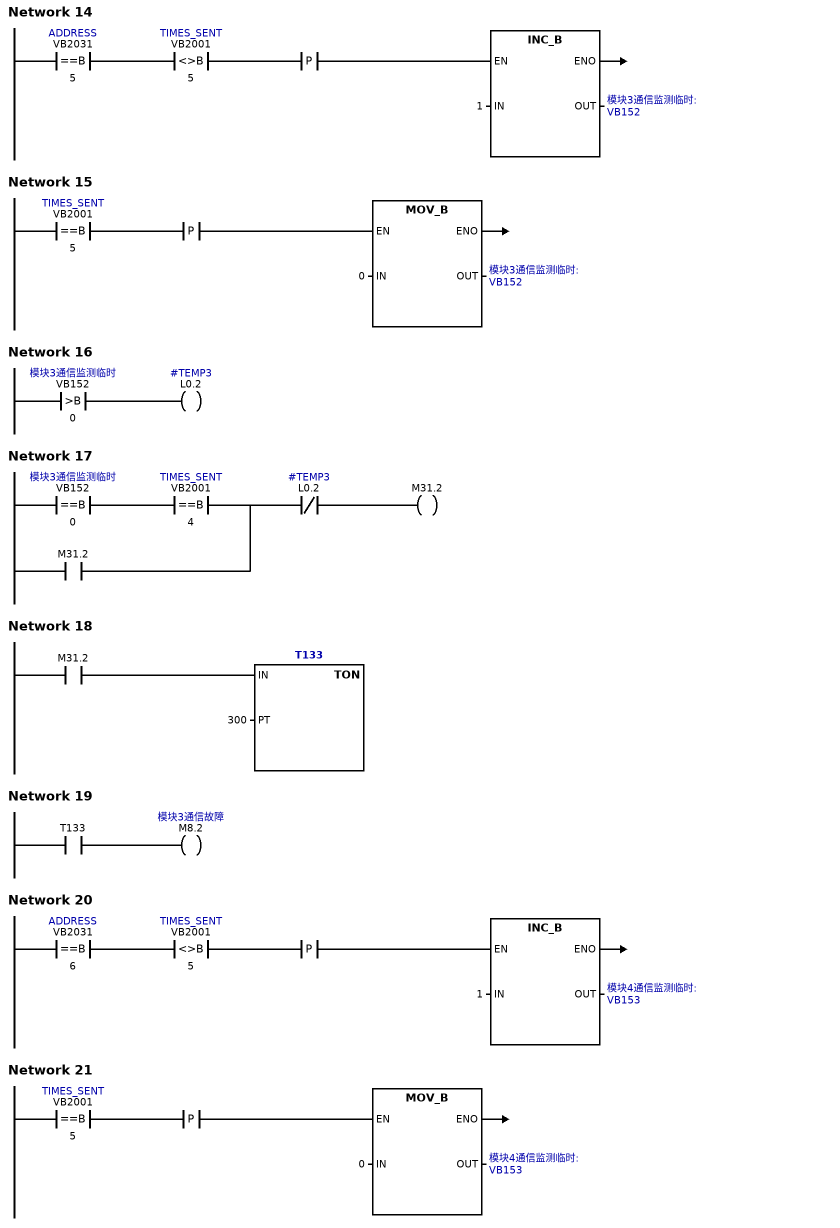
[picture p48: SBR53 networks 14-21]
Network 14
LDB=   ADDRESS:VB2031, 5
AB<>   TIMES_SENT:VB2001, 5
EU
MOVB   1, 模块3通信监测临时:VB152
INCB   模块3通信监测临时:VB152
Network 15
LDB=   TIMES_SENT:VB2001, 5
EU
MOVB   0, 模块3通信监测临时:VB152
Network 16
LDB>   模块3通信监测临时:VB152, 0
=      #TEMP3:L0.2
Network 17
LDB=   模块3通信监测临时:VB152, 0
AB=    TIMES_SENT:VB2001, 4
O      M31.2
AN     #TEMP3:L0.2
=      M31.2
Network 18
LD     M31.2
TON    T133, 300
Network 19
LD     T133
=      模块3通信故障:M8.2
Network 20
LDB=   ADDRESS:VB2031, 6
AB<>   TIMES_SENT:VB2001, 5
EU
MOVB   1, 模块4通信监测临时:VB153
INCB   模块4通信监测临时:VB153
Network 21
LDB=   TIMES_SENT:VB2001, 5
EU
MOVB   0, 模块4通信监测临时:VB153
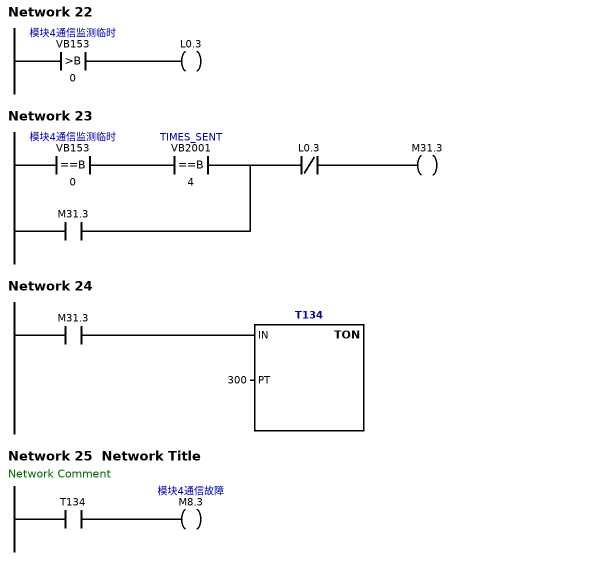
Network 22
LDB>   模块4通信监测临时:VB153, 0
=      L0.3
Network 23
LDB=   模块4通信监测临时:VB153, 0
AB=    TIMES_SENT:VB2001, 4
O      M31.3
AN     L0.3
=      M31.3
Network 24
LD     M31.3
TON    T134, 300
Network 25 // Network Title
// Network Comment
LD     T134
=      模块4通信故障:M8.3
END_SUBROUTINE_BLOCK

SUBROUTINE_BLOCK COMM_ARRAY:SBR54
TITLE=SUBROUTINE COMMENTS
VAR_INPUT
SLAVER_ADR:BYTE;	// LB0 
STAR_REG:BYTE;	// LB1 
REG_LEN:BYTE;	// LB2 
END_VAR
VAR_OUTPUT
ARRAY_T1:WORD;	// LW3 
ARRAY_T2:WORD;	// LW5 
ARRAY_T3:WORD;	// LW7 
ARRAY_T4:WORD;	// LW9 
END_VAR
BEGIN
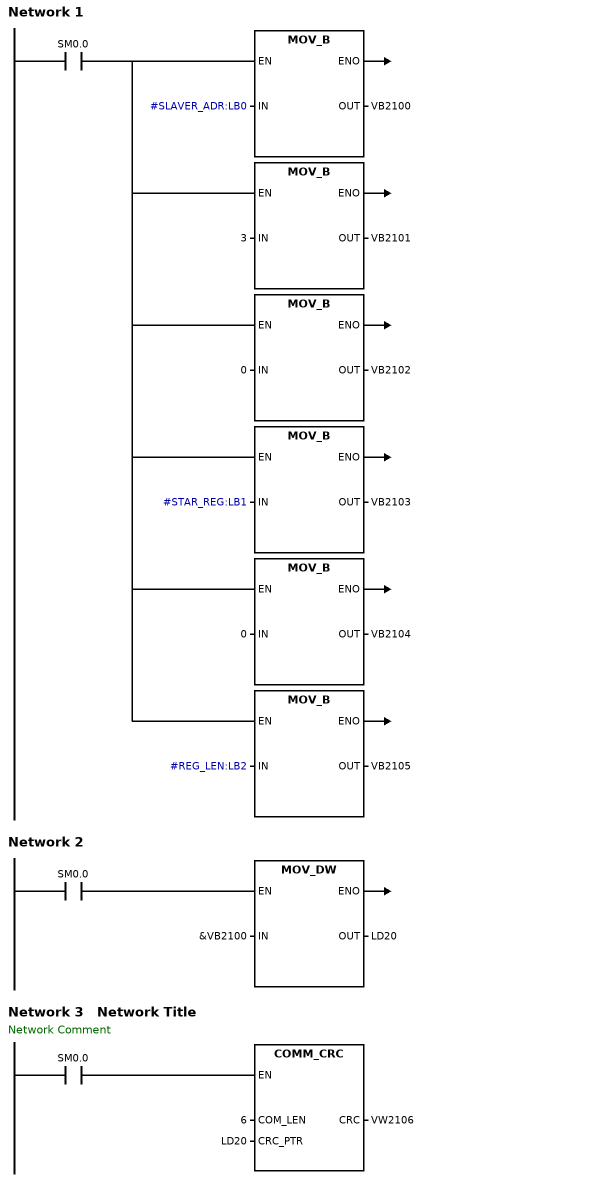
Network 1
LD     SM0.0
MOVB   #SLAVER_ADR:LB0, VB2100
MOVB   3, VB2101
MOVB   0, VB2102
MOVB   #STAR_REG:LB1, VB2103
MOVB   0, VB2104
MOVB   #REG_LEN:LB2, VB2105
Network 2
LD     SM0.0
MOVD   &VB2100, LD20
Network 3 //  Network Title
//  Network Comment
LD     SM0.0
CALL   COMM_CRC:SBR51, 6, LD20, VW2106
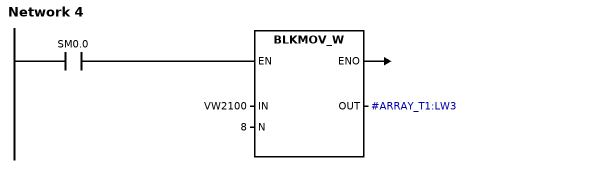
Network 4
LD     SM0.0
BMW    VW2100, #ARRAY_T1:LW3, 8
END_SUBROUTINE_BLOCK

// SBR55: protected block, not included

SUBROUTINE_BLOCK MES_SEND:SBR56
TITLE=SUBROUTINE COMMENTS
BEGIN
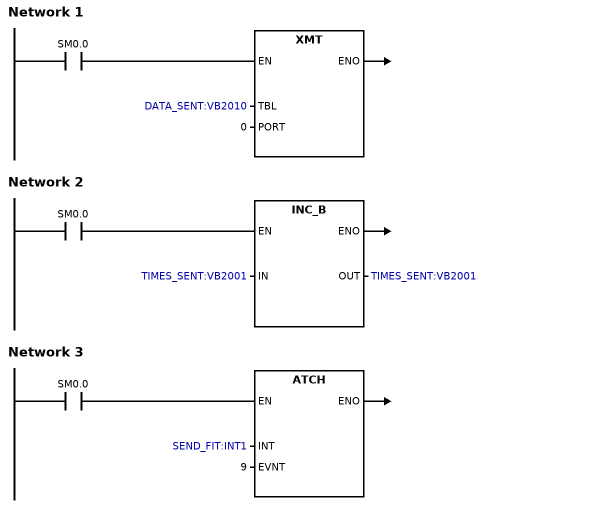
Network 1 // 
	
LD     SM0.0
XMT    DATA_SENT:VB2010, 0
Network 2
LD     SM0.0
INCB   TIMES_SENT:VB2001
Network 3
LD     SM0.0
ATCH   SEND_FIT:INT1, 9
Network 4 // Network Title
// Network Comment
END_SUBROUTINE_BLOCK

SUBROUTINE_BLOCK ARRAY_INSTR:SBR60
TITLE=旧的4块镇流器监测模块的地址分别是1,2,3,5
BEGIN
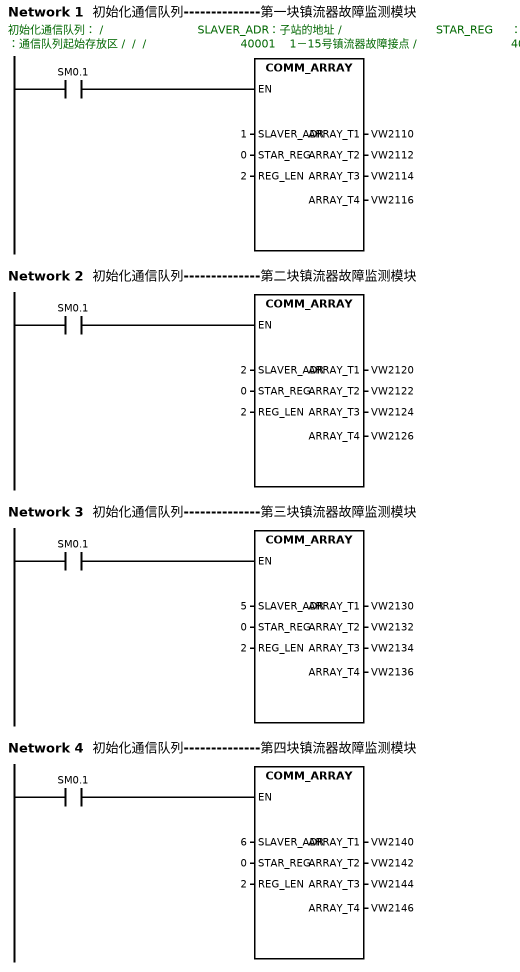
Network 1 // 初始化通信队列--------------第一块镇流器故障监测模块
// 初始化通信队列：
//                           SLAVER_ADR：子站的地址
//                           STAR_REG     ：子站数据起始寄存器
//                           REG_LEN        ：读取的数据寄存器长度
//                           ARRAY_T        ：通信队列起始存放区
// 
// 
//                           40001		1－15号镇流器故障接点
//                           40002		16－30号镇流器故障接点
//                         
LD     SM0.1
CALL   COMM_ARRAY:SBR54, 1, 0, 2, VW2110, VW2112, VW2114, VW2116
Network 2 // 初始化通信队列--------------第二块镇流器故障监测模块
LD     SM0.1
CALL   COMM_ARRAY:SBR54, 2, 0, 2, VW2120, VW2122, VW2124, VW2126
Network 3 // 初始化通信队列--------------第三块镇流器故障监测模块
LD     SM0.1
CALL   COMM_ARRAY:SBR54, 5, 0, 2, VW2130, VW2132, VW2134, VW2136
Network 4 // 初始化通信队列--------------第四块镇流器故障监测模块
LD     SM0.1
CALL   COMM_ARRAY:SBR54, 6, 0, 2, VW2140, VW2142, VW2144, VW2146
END_SUBROUTINE_BLOCK

// INT0: protected block, not included

INTERRUPT_BLOCK SEND_FIT:INT1
TITLE=
BEGIN
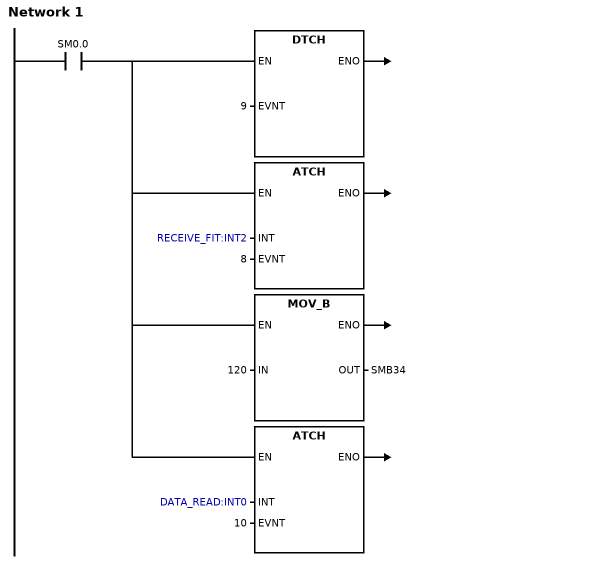
Network 1
LD     SM0.0
DTCH   9
ATCH   RECEIVE_FIT:INT2, 8
MOVB   120, SMB34
ATCH   DATA_READ:INT0, 10
END_INTERRUPT_BLOCK

// INT2: protected block, not included
